{attribute 'GeneratedUsingTerminal: EJ5151-0000-0016'}
{attribute addProperty BoxType "EJ5151-0000-0016"}
{attribute addProperty Id "Period_valueAT %I*UDINT4"}
{attribute addProperty CRC "615922771"}
{attribute addProperty Size "4"}
TYPE ENC_Inputs_24B63C53 EXTENDS InputBase_8311D824 :
STRUCT
	{attribute addProperty Name "Period_value"}
	Period_value AT %I* : UDINT;
END_STRUCT
END_TYPE

(* stored: Version 1.2.0.0, ProductVersion 3.1.4024.11
   DUT ENC_Inputs_24B63C53: Id {d45b8cde-005c-4f65-b09f-b878634fdcd5} *)
